// TIA Portal V18 export
DATA_BLOCK "Data_block_1"   // DB2
{ S7_Optimized_Access := 'TRUE' }
VERSION : 0.1
// stored: AutoNumber true, DBAccessibleFromOPCUA true, IsOnlyStoredInLoadMemory false, IsRetainMemResEnabled false, IsWriteProtectedInAS false, MemoryReserve 100
   VAR
      test : Bool;
   END_VAR
BEGIN
END_DATA_BLOCK
